TYPE ST_MCHMICommonData :
STRUCT
	bChangePage				: BOOL; //zmiana strony menu głównego
	wsActualState			: WSTRING;
	wsActualMode			: WSTRING;
	
	
END_STRUCT
END_TYPE

(* stored: Version 1.1.0.1
   DUT ST_MCHMICommonData: Id {480c357b-a090-08bb-2a3c-966a23f77842} *)
